(* PLC project TEST.project, CODESYS CODESYS V3.5 SP3 Patch 7 *)
(* stored: creationDateTime 2013-12-18T18:57:06.7863721, modificationDateTime 2013-12-18T18:56:49.0513577 *)

FUNCTION_BLOCK Drehkranz
  VAR
    Motor : INT;
    links : INT;
    rechts : INT;
    Endlagenschalter : BOOL;
    Endlagenschlater : INT;
  END_VAR

INITIAL_STEP Drehkranz steht:
END_STEP
TRANSITION FROM Drehkranz steht TO dreht links
  := Motor links;
END_TRANSITION
TRANSITION FROM Drehkranz steht TO dreht rechts
  := Motor rechts;
END_TRANSITION
STEP dreht links:
END_STEP
TRANSITION FROM dreht links TO Init
  := Endlagenschalter 8;
END_TRANSITION
STEP dreht rechts:
END_STEP
TRANSITION FROM dreht rechts TO Init
  := Endlagenschlater 9;
END_TRANSITION
END_FUNCTION_BLOCK
